// Mitsubishi GX Works2 project: 수위제어이상판단   PLC: Q02/Q02H

PROGRAM MAIN
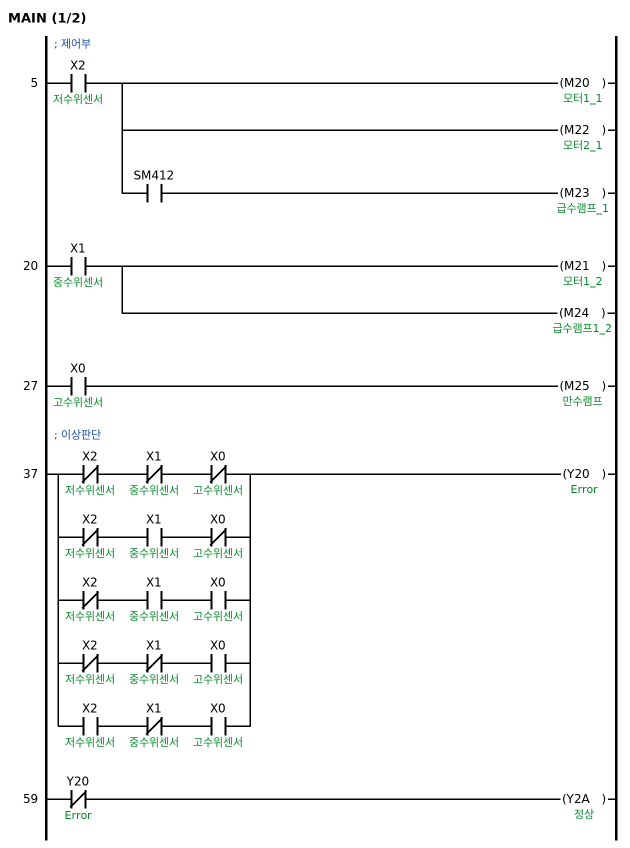
; 제어부
5     LD      X2  ; 저수위센서
      OUT     M20  ; 모터1_1
        [note] 
      OUT     M22  ; 모터2_1
        [note] 모터2_1
      AND     SM412
      OUT     M23  ; 급수램프_1
        [note] 
20    LD      X1  ; 중수위센서
      OUT     M21  ; 모터1_2
        [note] 
      OUT     M24  ; 급수램프1_2
        [note] 
27    LD      X0  ; 고수위센서
      OUT     M25  ; 만수램프
        [note] 
; 이상판단
37    LDI     X2  ; 저수위센서
      ANI     X1  ; 중수위센서
      ANI     X0  ; 고수위센서
      LDI     X2  ; 저수위센서
      AND     X1  ; 중수위센서
      ANI     X0  ; 고수위센서
      ORB
      LDI     X2  ; 저수위센서
      AND     X1  ; 중수위센서
      AND     X0  ; 고수위센서
      ORB
      LDI     X2  ; 저수위센서
      ANI     X1  ; 중수위센서
      AND     X0  ; 고수위센서
      ORB
      LD      X2  ; 저수위센서
      ANI     X1  ; 중수위센서
      AND     X0  ; 고수위센서
      ORB
      OUT     Y20  ; Error
        [note] 
59    LDI     Y20  ; Error
      OUT     Y2A  ; 정상
        [note] 
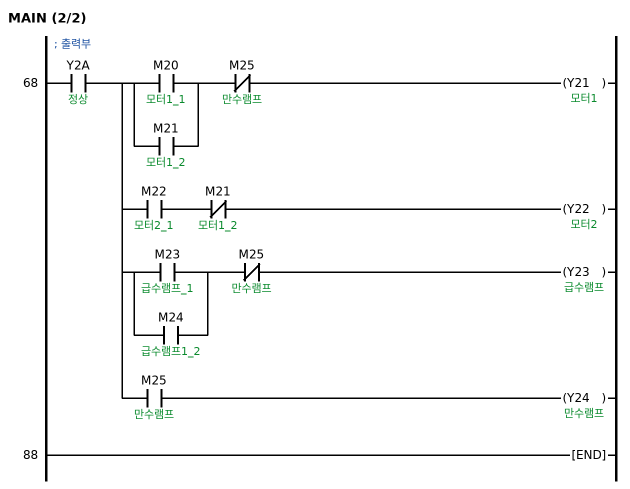
; 출력부
68    LD      Y2A  ; 정상
      MPS
      LD      M20  ; 모터1_1
      OR      M21  ; 모터1_2
      ANB
      ANI     M25  ; 만수램프
      OUT     Y21  ; 모터1
      MRD
      AND     M22  ; 모터2_1
      ANI     M21  ; 모터1_2
      OUT     Y22  ; 모터2
      MRD
      LD      M23  ; 급수램프_1
      OR      M24  ; 급수램프1_2
      ANB
      ANI     M25  ; 만수램프
      OUT     Y23  ; 급수램프
      MPP
      AND     M25  ; 만수램프
      OUT     Y24  ; 만수램프
88    END
END_PROGRAM

// device comments not shown above
M0  ; 보조0
M1  ; 보조1
M2  ; 보조2
M3  ; 보조3
